{attribute 'linkalways'}
{attribute 'no_explicit_call' := 'do not call this POU directly'}
FUNCTION_BLOCK InstanceAddedEvent EXTENDS Event IMPLEMENTS I_InstanceAddedEvent
VAR
	_instance : I_Instance;
END_VAR

PROPERTY PUBLIC Instance : I_Instance
GET
Instance := _instance;
END_GET
END_PROPERTY

METHOD PUBLIC Notify
VAR_INPUT
	Instance : I_Instance;
END_VAR
_instance := Instance;
NotifySubscribers();
END_METHOD

END_FUNCTION_BLOCK

(* stored: Version 1.1.0.1, ProductVersion 3.1.4024.11
   POU InstanceAddedEvent: Id {a53b82ca-f1dc-446c-adff-ccbf595d3c87}, SpecialFunc None
   Property Instance: Id {809619db-ec1f-4cf6-bf24-66d43aeb16d2}
   Get Get: Id {bc678033-c666-4ceb-bc8f-37cf9fee58ea}
   Method Notify: Id {24509aef-7228-4a5e-9e32-fa2674861881} *)
